FUNCTION_BLOCK FB_Regulator
VAR_INPUT
	iI: INT;
	lrVelocity	:	LREAL := 360;
END_VAR
VAR_OUTPUT
q_asResult: ARRAY [1..20] OF STRING;
q_xError	:	BOOL;
END_VAR
VAR_IN_OUT
	iq_stRegulator	:	ST_Regulator;
END_VAR
VAR
	

mcPower	:	MC_Power;
mcSetHome	:	MC_SetPosition;
mcReset	:	MC_Reset;
mcMoveAbsolute : ARRAY[1..2] OF MC_MoveAbsolute;
mcStatus : MC_ReadStatus;

mcHalt	:	MC_Halt;

	iPressDiff: INT;
	iTolerance: INT := 50;
	xMoveOK: BOOL;
	iStep: INT;
	
	indexResult: INT := 1;
	
	xInitComplete	:	BOOL := FALSE;
	
	ftBackToAuto	:	F_TRIG;
	iPercSPOld: UINT;
	imcBlockIndex: INT;
	imcBlockIndexPrev : INT;
	
	rtEnable : R_TRIG;
END_VAR

(* Regulator Function Block *)
(* Alex Wallace, 2014-10-16 *)
(* Modified in 2.5.3 to remove all pressure SP  based code *)

rtEnable(CLK:=iq_stRegulator.xRegEnab);

(* Regulator Pressure Calculation *)
iq_stRegulator.wInPress := LIMIT(0, F_rPressure(iRawVoltage := iq_stRegulator.i_iRawInPress), 10000);
iq_stRegulator.wOutPress := LIMIT(0, F_rPressure(iRawVoltage := iq_stRegulator.i_iRawOutPress), 10000);


(* Basic regulator interlocking *)


(* Check for regulator enable *)
xMoveOK := iq_stRegulator.xRegEnab;
IF NOT xMoveOK THEN
	(*iq_stRegulator.wPressSP := 0; not preferred *)
	iq_stRegulator.xRegEnab := FALSE;
	(* add motor error here *)
END_IF

IF q_xError THEN
	iStep := 9000;
ELSIF rtEnable.Q THEN
	xInitComplete := FALSE;
	iStep := 10;
ELSIF xInitComplete THEN
	iStep := 3000;
END_IF


CASE iStep OF
	0: iStep := 10;
	10:
	(* Start by initializing the motor axis *)
	mcPower.Enable := TRUE;
	iq_stRegulator.lrUpperLimPos := 2887;
	IF mcPower.Status THEN
		xInitComplete := TRUE;
		q_asResult[indexResult] := 'Motor init success';
		indexResult := indexResult + 1;
		iStep := 3000;
	ELSIF mcPower.Error THEN
		mcPower.Enable := FALSE;
		iStep := 9000;
		q_xError	:=	TRUE;
		q_asResult[indexResult] := CONCAT('Initilizing regulator motor in step 10 failed with error code: ', UDINT_TO_STRING(mcPower.ErrorID));
		indexResult := indexResult +1;
	END_IF
		
	//Knob controls
	3000:
	
	IF iq_stRegulator.i_iPercSP <> iPercSPOld  AND xMoveOK THEN
		mcMoveAbsolute[imcBlockIndex].Execute := FALSE;
		imcBlockIndex := imcBlockIndex + 1;
		IF imcBlockIndex >2 THEN imcBlockIndex := 1; END_IF
		mcMoveAbsolute[imcBlockIndex].Position := LIMIT(0, UINT_TO_LREAL(iq_stRegulator.i_iPercSP) * iq_stRegulator.lrUpperLimPos/65535, MAX(iq_stRegulator.lrUpperLimPos,1));
		mcMoveAbsolute[imcBlockIndex].Execute := TRUE;
		iPercSPOld := iq_stRegulator.i_iPercSP;
	ELSIF mcMoveAbsolute[imcBlockIndex].Done or mcMoveAbsolute[imcBlockIndex].CommandAborted or mcMoveAbsolute[imcBlockIndex].Busy or mcMoveAbsolute[imcBlockIndex].Error THEN
		mcMoveAbsolute[imcBlockIndex].Execute := FALSE;
	END_IF
	
	9000:
	(* Error *)
	mcReset.Execute := iq_stRegulator.xRegEnab;
	IF mcReset.Done THEN
		q_xError := FALSE;
		mcReset.Execute := FALSE;
		iStep:=10;
	END_IF
	
END_CASE

//Reset the debugging index
IF indexResult > 20 THEN indexResult := 1; END_IF

(* Regulator Percentage Open *)
(* Calculate the regulator percentage open, based on 6.5 turns to fully open *)

iq_stRegulator.wPercentageOpen := LREAL_TO_WORD( (iq_stRegulator.stRegulatorMotor.NcToPlc.ActPos / MAX(iq_stRegulator.lrUpperLimPos,1))*100);

(* Run the mc blocks *)
iq_stRegulator.stRegulatorMotor();
ActPower();

mcSetHome(Execute:=NOT(iq_stRegulator.xRegLoLS) AND iq_stRegulator.stRegulatorMotor.Status.StandStill, Axis:=iq_stRegulator.stRegulatorMotor, Position:=0, Mode:=FALSE);
IF NOT iq_stRegulator.xRegHiLS THEN iq_stRegulator.lrUpperLimPos := iq_stRegulator.stRegulatorMotor.NcToPlc.ActPos; END_IF
mcReset(Axis:=iq_stRegulator.stRegulatorMotor);

FOR iI := 1 TO 2 DO
mcMoveAbsolute[iI](Axis := iq_stRegulator.stRegulatorMotor, Velocity:=iq_stRegulator.lrVelocity, BufferMode:=MC_Aborting);
END_FOR

IF mcMoveAbsolute[1].Error OR mcMoveAbsolute[2].Error THEN
	q_xError	:=	TRUE;
	mcMoveAbsolute[1].Execute := FALSE;
	mcMoveAbsolute[2].Execute := FALSE;
	q_asResult[indexResult] := 'Error occured with motion blocks';
	indexResult := indexResult +1;
ELSIF mcPower.Error THEN
	q_xError := TRUE;
	q_asResult[indexResult] := concat('mcPower block error: ', UDINT_TO_STRING(mcPower.ErrorID));
END_IF

ACTION ActPower:
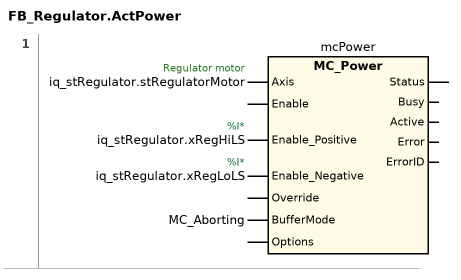
// NETWORK 1
//   iq_stRegulator.stRegulatorMotor: Regulator motor
//   iq_stRegulator.xRegHiLS: AT %I*
//   iq_stRegulator.xRegLoLS: AT %I*
mcPower(
    Axis := iq_stRegulator.stRegulatorMotor,
    Enable_Positive := iq_stRegulator.xRegHiLS,
    Enable_Negative := iq_stRegulator.xRegLoLS,
    BufferMode := MC_Aborting); // MC_Power
END_ACTION

END_FUNCTION_BLOCK

(* stored: Version 1.1.0.1, ProductVersion 3.1.4018.5
   POU FB_Regulator: Id {aa85a243-cf4d-4b77-a154-ab7f2bb33020}, SpecialFunc None
   Action ActPower: Id {e34cb278-3582-4d00-9245-81999faf4464} *)
